(* PLC project PLC, Beckhoff Automation GmbH TwinCAT PLC Control 3.5.20.60 *)
(* stored: creationDateTime 2026-07-21T08:44:24.682903, modificationDateTime 2026-07-21T08:44:24.682903 *)

TYPE ST_ADS_API_ScadaViewerApp_PLC_In_Status :

STRUCT

	Heartbeat			:	BOOL;	// |1| Heartbeat signál
	Ready				:	BOOL;	// |2| Aplikace připravena na činnost
	
END_STRUCT

END_TYPE
